Staubli VAL3: setCmdPos.pgx

program setCmdPos(num x_nAxisNum (dimensions=1))
  local num l_nCurrentPos
  local num l_nCmdPos
begin
  //把当前位置赋给驱动器
  l_nCurrentPos=aioGet(aiPosFbk[x_nAxisNum])
  aioSet(aoPosCmd[x_nAxisNum],l_nCurrentPos)
end
